SYSTEM test
  (* Version 1.0, 2023-02-17, Franz *)
  APPLICATION testApp
  END_APPLICATION
  DEVICE FORTE_PC : FORTE_PC(MGR_ID := "192.168.4.1:61499")
    {SET_ATTRIBUTE(Profile, HOLOBLOC)}
    RESOURCE EMB_RES : EMB_RES
    END_RESOURCE
  END_DEVICE
  SEGMENTS
    Ethernet : Ethernet;
  END_SEGMENTS
  LINKS
    FORTE_PC => Ethernet;
  END_LINKS
END_SYSTEM
